TYPE TO_Cam_Struct_PointData :
STRUCT
	x: LREAL;
	y:LREAL;

END_STRUCT
END_TYPE

(* stored: Version 1.1.0.1
   DUT TO_Cam_Struct_PointData: Id {b824af2f-2b79-4445-858a-f88b06b9c75e} *)
